Universal Robots PolyScope program: L01_movejlp.urp

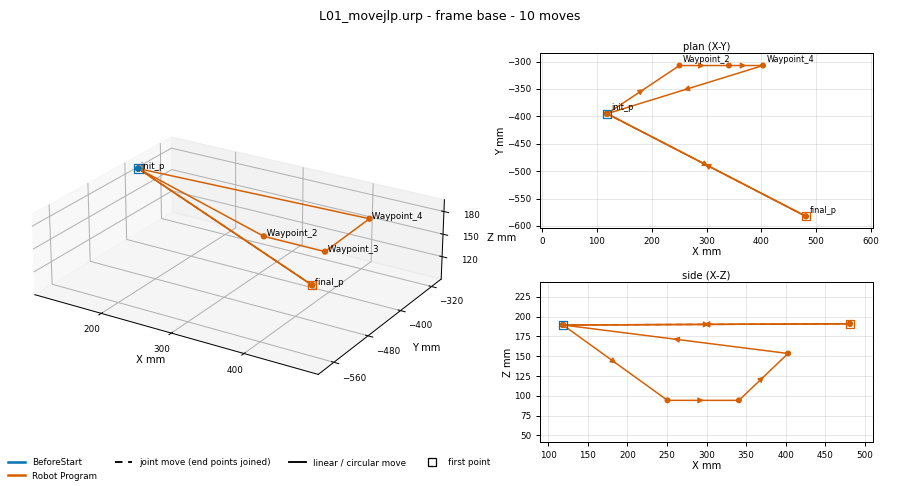
[picture p0: tool path of L01_movejlp.urp in frame base, 10 of 10 moves have a stored position in this frame; points joined in program order, loops and branches not executed]
Program L01_movejlp (installation=default directory=/programs createdIn=5.9.1.1031110 lastSavedIn=5.9.1.1031110 robotSerialNumber=20195501059)
Calibrated DH parameters: a=[0.000146, -0.418764, -0.053981, 0.000058, -0.000023, 0]; d=[0.162545, 37.319448, -206.067439, 168.881546, 0.09955, 0.099464]; alpha=[1.57004, -0.001979, 0.002304, 1.570607, -1.57066, 0]; deltaTheta=[0, -0.174616, -1.258233, 1.432844, -0.000001, 0]
BeforeStart
  URCap Gripper Activate (Robotiq_Grippers, Robotiq Inc.) dataModel(ResetAndActivateKey=false)
  URCap Gripper (Robotiq_Grippers, Robotiq Inc.) dataModel(position=100.0, force=100.0, speed=100.0, positionInDouble=100.0, forceInDouble=100.0, speedInDouble=100.0, slaveIds=[9], blocking=true)
  MoveJ speed 60 deg/s, acceleration 80 deg/s^2 (useActiveTCP=true) feature=Base
    Waypoint init_p: TCP in base x=118.516 y=-395.223 z=189.498 mm, rx=2.271 ry=1.6279 rz=-0.3642 rad; joints [88.026, -113.926, 136.576, -136.365, 269.786, 106.722] deg; TCP offset x=0 y=0 z=174 mm, rx=0 ry=0 rz=0 rad
Robot Program (runOnlyOnce=true)
  MoveJ speed 60 deg/s, acceleration 80 deg/s^2 (useActiveTCP=true) feature=Base
    Waypoint final_p: TCP in base x=481.277 y=-582.487 z=191.042 mm, rx=2.3645 ry=1.2104 rz=0.4255 rad; joints [112.273, -66.723, 92.652, -141.3, 289.391, 152.475] deg
    Waypoint init_p: TCP in base x=118.516 y=-395.223 z=189.498 mm, rx=2.271 ry=1.6279 rz=-0.3642 rad; joints [88.026, -113.926, 136.576, -136.365, 269.786, 106.722] deg
  MoveL speed 250 mm/s, acceleration 1200 mm/s^2 (useActiveTCP=true) feature=Base
    Waypoint final_p: TCP in base x=481.277 y=-582.487 z=191.042 mm, rx=2.3645 ry=1.2104 rz=0.4255 rad; joints [112.273, -66.723, 92.652, -141.3, 289.391, 152.475] deg
    Waypoint init_p: TCP in base x=118.516 y=-395.223 z=189.498 mm, rx=2.271 ry=1.6279 rz=-0.3642 rad; joints [88.026, -113.926, 136.576, -136.365, 269.786, 106.722] deg
  Loop Counting (count=3) loopVariable(name=Loop_1)
    MoveP speed 250 mm/s, acceleration 800 mm/s^2 (blendRadius=0.025 useActiveTCP=true) feature=Base
      Waypoint Waypoint_2: TCP in base x=250.609 y=-307.341 z=94.3 mm, rx=-2.2211 ry=-2.2047 rz=-0.0018 rad; joints [109.681, -96.819, 130.14, -122.661, 269.843, 110.127] deg
      Waypoint Waypoint_3: TCP in base x=340.834 y=-307.333 z=94.285 mm, rx=-2.2211 ry=-2.2047 rz=-0.0017 rad; joints [121.089, -87.728, 121.516, -123.093, 269.957, 121.539] deg
      Waypoint Waypoint_4: TCP in base x=402.984 y=-307.32 z=153.537 mm, rx=-2.2211 ry=-2.2047 rz=-0.0017 rad; joints [127.389, -85.481, 109.233, -113.048, 270.009, 127.825] deg
      Waypoint init_p: TCP in base x=118.516 y=-395.223 z=189.498 mm, rx=2.271 ry=1.6279 rz=-0.3642 rad; joints [88.026, -113.926, 136.576, -136.365, 269.786, 106.722] deg
  MoveL speed 250 mm/s, acceleration 1200 mm/s^2 (useActiveTCP=true) feature=Base
    Waypoint init_p: TCP in base x=118.516 y=-395.223 z=189.498 mm, rx=2.271 ry=1.6279 rz=-0.3642 rad; joints [88.026, -113.926, 136.576, -136.365, 269.786, 106.722] deg
